Staubli VAL3: RobotCommand.pjx

--- RobotCommand.pjx ---
Parameters version=s7.7.2 stackSize=5000 millimeterUnit=true
Program file=start.pgx
Program file=stop.pgx
Data file=RobotCommand.dtx

--- RobotCommand.dtx ---
public bool bIsValid = false
public num nMode
public num nRemoteCtrlPeriod
public num nMotionCmdType
public num nMotionCmdData[6]
public bool nDigitalOutputs[16]
public num nAnalogOutputs[4]
